# EPICS substitutions: db/valve.substitutions
# valve substituion file

file db/valve.db {
  pattern { V }
    { V1 }
    { V2 }
}
